KUKA KRL program: Sps1.sub

&ACCESS RV
&PARAM TPVW_VERSION=8.3.18
DEF  SPS1 ( )
; FOLD ;%{H} %MKUKATPVW
;Init part of vw_usr_s
VW_USR_S (#USR_INIT_SUB1)

LOOP
;Freilaufende SPS
MAKROSUBMIT1()

WAIT FOR NOT $POWER_FAIL
ENDLOOP
END
;ENDFOLD
